// TIA Portal V20 export
ORGANIZATION_BLOCK "7000_Main"   // OB127, LAD, ProgramCycle
TITLE = "Main Program Sweep (Cycle)"
// stored: SetENOAutomatically false
   VAR_INPUT
      Initial_Call : Bool;   // Initial call of this OB
      Remanence : Bool;   // =True, if remanent data are available
   END_VAR
BEGIN

REGION Network 1: 2201_StackCalculate
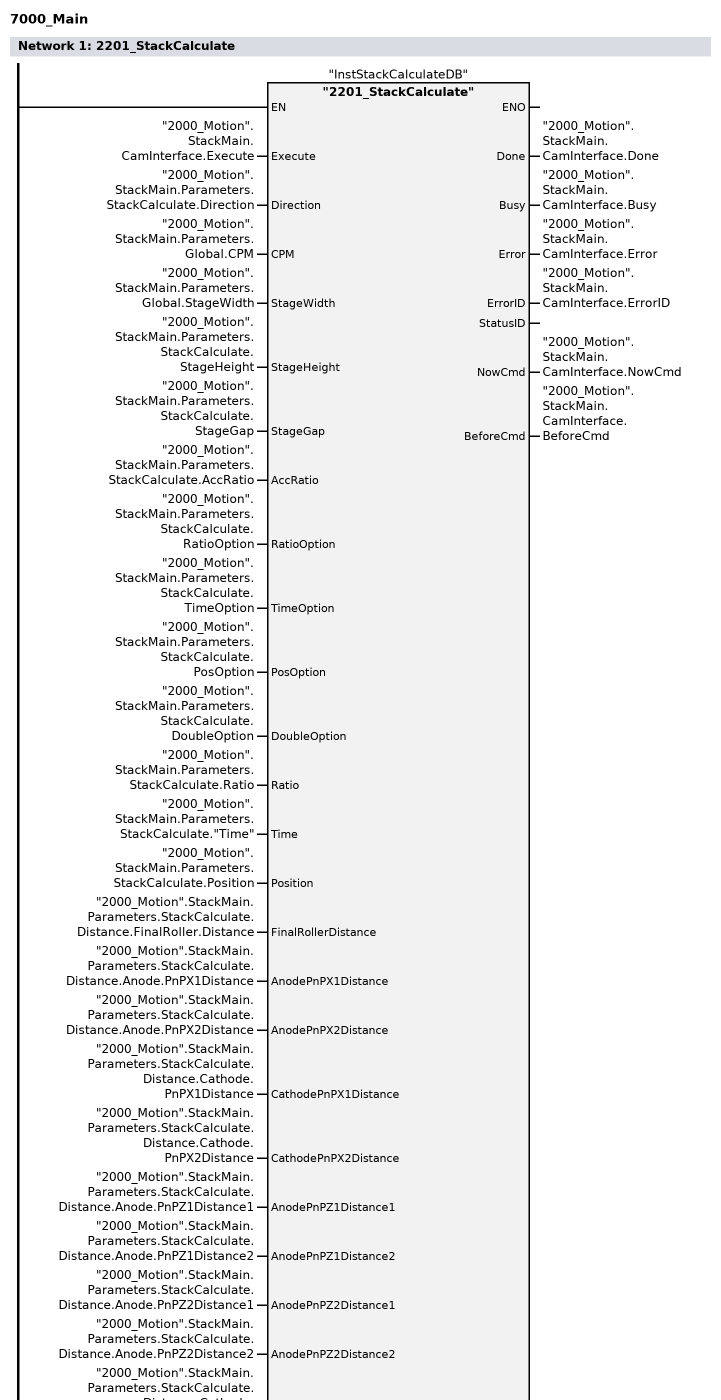
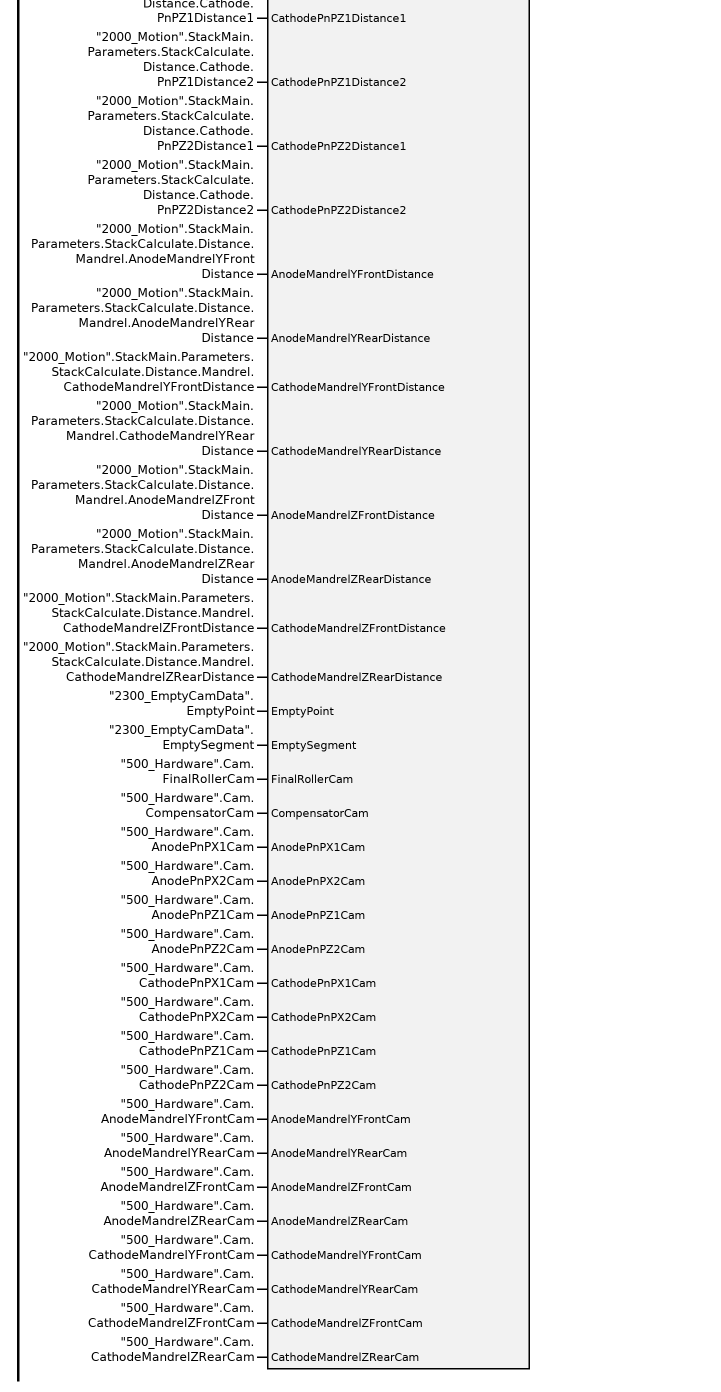
   RUNG wire#powerrail
      "InstStackCalculateDB"(Execute := "2000_Motion".StackMain.CamInterface.Execute, Direction := "2000_Motion".StackMain.Parameters.StackCalculate.Direction, CPM := "2000_Motion".StackMain.Parameters.Global.CPM, StageWidth := "2000_Motion".StackMain.Parameters.Global.StageWidth, StageHeight := "2000_Motion".StackMain.Parameters.StackCalculate.StageHeight, StageGap := "2000_Motion".StackMain.Parameters.StackCalculate.StageGap, AccRatio := "2000_Motion".StackMain.Parameters.StackCalculate.AccRatio, RatioOption := "2000_Motion".StackMain.Parameters.StackCalculate.RatioOption, TimeOption := "2000_Motion".StackMain.Parameters.StackCalculate.TimeOption, PosOption := "2000_Motion".StackMain.Parameters.StackCalculate.PosOption, DoubleOption := "2000_Motion".StackMain.Parameters.StackCalculate.DoubleOption, Ratio := "2000_Motion".StackMain.Parameters.StackCalculate.Ratio, "Time" := "2000_Motion".StackMain.Parameters.StackCalculate."Time", Position := "2000_Motion".StackMain.Parameters.StackCalculate.Position, FinalRollerDistance := "2000_Motion".StackMain.Parameters.StackCalculate.Distance.FinalRoller.Distance, AnodePnPX1Distance := "2000_Motion".StackMain.Parameters.StackCalculate.Distance.Anode.PnPX1Distance, AnodePnPX2Distance := "2000_Motion".StackMain.Parameters.StackCalculate.Distance.Anode.PnPX2Distance, CathodePnPX1Distance := "2000_Motion".StackMain.Parameters.StackCalculate.Distance.Cathode.PnPX1Distance, CathodePnPX2Distance := "2000_Motion".StackMain.Parameters.StackCalculate.Distance.Cathode.PnPX2Distance, AnodePnPZ1Distance1 := "2000_Motion".StackMain.Parameters.StackCalculate.Distance.Anode.PnPZ1Distance1, AnodePnPZ1Distance2 := "2000_Motion".StackMain.Parameters.StackCalculate.Distance.Anode.PnPZ1Distance2, AnodePnPZ2Distance1 := "2000_Motion".StackMain.Parameters.StackCalculate.Distance.Anode.PnPZ2Distance1, AnodePnPZ2Distance2 := "2000_Motion".StackMain.Parameters.StackCalculate.Distance.Anode.PnPZ2Distance2, CathodePnPZ1Distance1 := "2000_Motion".StackMain.Parameters.StackCalculate.Distance.Cathode.PnPZ1Distance1, CathodePnPZ1Distance2 := "2000_Motion".StackMain.Parameters.StackCalculate.Distance.Cathode.PnPZ1Distance2, CathodePnPZ2Distance1 := "2000_Motion".StackMain.Parameters.StackCalculate.Distance.Cathode.PnPZ2Distance1, CathodePnPZ2Distance2 := "2000_Motion".StackMain.Parameters.StackCalculate.Distance.Cathode.PnPZ2Distance2, AnodeMandrelYFrontDistance := "2000_Motion".StackMain.Parameters.StackCalculate.Distance.Mandrel.AnodeMandrelYFrontDistance, AnodeMandrelYRearDistance := "2000_Motion".StackMain.Parameters.StackCalculate.Distance.Mandrel.AnodeMandrelYRearDistance, CathodeMandrelYFrontDistance := "2000_Motion".StackMain.Parameters.StackCalculate.Distance.Mandrel.CathodeMandrelYFrontDistance, CathodeMandrelYRearDistance := "2000_Motion".StackMain.Parameters.StackCalculate.Distance.Mandrel.CathodeMandrelYRearDistance, AnodeMandrelZFrontDistance := "2000_Motion".StackMain.Parameters.StackCalculate.Distance.Mandrel.AnodeMandrelZFrontDistance, AnodeMandrelZRearDistance := "2000_Motion".StackMain.Parameters.StackCalculate.Distance.Mandrel.AnodeMandrelZRearDistance, CathodeMandrelZFrontDistance := "2000_Motion".StackMain.Parameters.StackCalculate.Distance.Mandrel.CathodeMandrelZFrontDistance, CathodeMandrelZRearDistance := "2000_Motion".StackMain.Parameters.StackCalculate.Distance.Mandrel.CathodeMandrelZRearDistance, EmptyPoint := "2300_EmptyCamData".EmptyPoint, EmptySegment := "2300_EmptyCamData".EmptySegment, FinalRollerCam := "500_Hardware".Cam.FinalRollerCam, CompensatorCam := "500_Hardware".Cam.CompensatorCam, AnodePnPX1Cam := "500_Hardware".Cam.AnodePnPX1Cam, AnodePnPX2Cam := "500_Hardware".Cam.AnodePnPX2Cam, AnodePnPZ1Cam := "500_Hardware".Cam.AnodePnPZ1Cam, AnodePnPZ2Cam := "500_Hardware".Cam.AnodePnPZ2Cam, CathodePnPX1Cam := "500_Hardware".Cam.CathodePnPX1Cam, CathodePnPX2Cam := "500_Hardware".Cam.CathodePnPX2Cam, CathodePnPZ1Cam := "500_Hardware".Cam.CathodePnPZ1Cam, CathodePnPZ2Cam := "500_Hardware".Cam.CathodePnPZ2Cam, AnodeMandrelYFrontCam := "500_Hardware".Cam.AnodeMandrelYFrontCam, AnodeMandrelYRearCam := "500_Hardware".Cam.AnodeMandrelYRearCam, AnodeMandrelZFrontCam := "500_Hardware".Cam.AnodeMandrelZFrontCam, AnodeMandrelZRearCam := "500_Hardware".Cam.AnodeMandrelZRearCam, CathodeMandrelYFrontCam := "500_Hardware".Cam.CathodeMandrelYFrontCam, CathodeMandrelYRearCam := "500_Hardware".Cam.CathodeMandrelYRearCam, CathodeMandrelZFrontCam := "500_Hardware".Cam.CathodeMandrelZFrontCam, CathodeMandrelZRearCam := "500_Hardware".Cam.CathodeMandrelZRearCam, Done => "2000_Motion".StackMain.CamInterface.Done, Busy => "2000_Motion".StackMain.CamInterface.Busy, Error => "2000_Motion".StackMain.CamInterface.Error, ErrorID => "2000_Motion".StackMain.CamInterface.ErrorID, NowCmd => "2000_Motion".StackMain.CamInterface.NowCmd, BeforeCmd => "2000_Motion".StackMain.CamInterface.BeforeCmd, StatusID =>)
   END_RUNG
   // the same network as SCL:
   "InstStackCalculateDB"(Execute := "2000_Motion".StackMain.CamInterface.Execute,   // "2201_StackCalculate"
                          Direction := "2000_Motion".StackMain.Parameters.StackCalculate.Direction,
                          CPM := "2000_Motion".StackMain.Parameters.Global.CPM,
                          StageWidth := "2000_Motion".StackMain.Parameters.Global.StageWidth,
                          StageHeight := "2000_Motion".StackMain.Parameters.StackCalculate.StageHeight,
                          StageGap := "2000_Motion".StackMain.Parameters.StackCalculate.StageGap,
                          AccRatio := "2000_Motion".StackMain.Parameters.StackCalculate.AccRatio,
                          RatioOption := "2000_Motion".StackMain.Parameters.StackCalculate.RatioOption,
                          TimeOption := "2000_Motion".StackMain.Parameters.StackCalculate.TimeOption,
                          PosOption := "2000_Motion".StackMain.Parameters.StackCalculate.PosOption,
                          DoubleOption := "2000_Motion".StackMain.Parameters.StackCalculate.DoubleOption,
                          Ratio := "2000_Motion".StackMain.Parameters.StackCalculate.Ratio,
                          "Time" := "2000_Motion".StackMain.Parameters.StackCalculate."Time",
                          Position := "2000_Motion".StackMain.Parameters.StackCalculate.Position,
                          FinalRollerDistance := "2000_Motion".StackMain.Parameters.StackCalculate.Distance.FinalRoller.Distance,
                          AnodePnPX1Distance := "2000_Motion".StackMain.Parameters.StackCalculate.Distance.Anode.PnPX1Distance,
                          AnodePnPX2Distance := "2000_Motion".StackMain.Parameters.StackCalculate.Distance.Anode.PnPX2Distance,
                          CathodePnPX1Distance := "2000_Motion".StackMain.Parameters.StackCalculate.Distance.Cathode.PnPX1Distance,
                          CathodePnPX2Distance := "2000_Motion".StackMain.Parameters.StackCalculate.Distance.Cathode.PnPX2Distance,
                          AnodePnPZ1Distance1 := "2000_Motion".StackMain.Parameters.StackCalculate.Distance.Anode.PnPZ1Distance1,
                          AnodePnPZ1Distance2 := "2000_Motion".StackMain.Parameters.StackCalculate.Distance.Anode.PnPZ1Distance2,
                          AnodePnPZ2Distance1 := "2000_Motion".StackMain.Parameters.StackCalculate.Distance.Anode.PnPZ2Distance1,
                          AnodePnPZ2Distance2 := "2000_Motion".StackMain.Parameters.StackCalculate.Distance.Anode.PnPZ2Distance2,
                          CathodePnPZ1Distance1 := "2000_Motion".StackMain.Parameters.StackCalculate.Distance.Cathode.PnPZ1Distance1,
                          CathodePnPZ1Distance2 := "2000_Motion".StackMain.Parameters.StackCalculate.Distance.Cathode.PnPZ1Distance2,
                          CathodePnPZ2Distance1 := "2000_Motion".StackMain.Parameters.StackCalculate.Distance.Cathode.PnPZ2Distance1,
                          CathodePnPZ2Distance2 := "2000_Motion".StackMain.Parameters.StackCalculate.Distance.Cathode.PnPZ2Distance2,
                          AnodeMandrelYFrontDistance := "2000_Motion".StackMain.Parameters.StackCalculate.Distance.Mandrel.AnodeMandrelYFrontDistance,
                          AnodeMandrelYRearDistance := "2000_Motion".StackMain.Parameters.StackCalculate.Distance.Mandrel.AnodeMandrelYRearDistance,
                          CathodeMandrelYFrontDistance := "2000_Motion".StackMain.Parameters.StackCalculate.Distance.Mandrel.CathodeMandrelYFrontDistance,
                          CathodeMandrelYRearDistance := "2000_Motion".StackMain.Parameters.StackCalculate.Distance.Mandrel.CathodeMandrelYRearDistance,
                          AnodeMandrelZFrontDistance := "2000_Motion".StackMain.Parameters.StackCalculate.Distance.Mandrel.AnodeMandrelZFrontDistance,
                          AnodeMandrelZRearDistance := "2000_Motion".StackMain.Parameters.StackCalculate.Distance.Mandrel.AnodeMandrelZRearDistance,
                          CathodeMandrelZFrontDistance := "2000_Motion".StackMain.Parameters.StackCalculate.Distance.Mandrel.CathodeMandrelZFrontDistance,
                          CathodeMandrelZRearDistance := "2000_Motion".StackMain.Parameters.StackCalculate.Distance.Mandrel.CathodeMandrelZRearDistance,
                          EmptyPoint := "2300_EmptyCamData".EmptyPoint,
                          EmptySegment := "2300_EmptyCamData".EmptySegment,
                          FinalRollerCam := "500_Hardware".Cam.FinalRollerCam,
                          CompensatorCam := "500_Hardware".Cam.CompensatorCam,
                          AnodePnPX1Cam := "500_Hardware".Cam.AnodePnPX1Cam,
                          AnodePnPX2Cam := "500_Hardware".Cam.AnodePnPX2Cam,
                          AnodePnPZ1Cam := "500_Hardware".Cam.AnodePnPZ1Cam,
                          AnodePnPZ2Cam := "500_Hardware".Cam.AnodePnPZ2Cam,
                          CathodePnPX1Cam := "500_Hardware".Cam.CathodePnPX1Cam,
                          CathodePnPX2Cam := "500_Hardware".Cam.CathodePnPX2Cam,
                          CathodePnPZ1Cam := "500_Hardware".Cam.CathodePnPZ1Cam,
                          CathodePnPZ2Cam := "500_Hardware".Cam.CathodePnPZ2Cam,
                          AnodeMandrelYFrontCam := "500_Hardware".Cam.AnodeMandrelYFrontCam,
                          AnodeMandrelYRearCam := "500_Hardware".Cam.AnodeMandrelYRearCam,
                          AnodeMandrelZFrontCam := "500_Hardware".Cam.AnodeMandrelZFrontCam,
                          AnodeMandrelZRearCam := "500_Hardware".Cam.AnodeMandrelZRearCam,
                          CathodeMandrelYFrontCam := "500_Hardware".Cam.CathodeMandrelYFrontCam,
                          CathodeMandrelYRearCam := "500_Hardware".Cam.CathodeMandrelYRearCam,
                          CathodeMandrelZFrontCam := "500_Hardware".Cam.CathodeMandrelZFrontCam,
                          CathodeMandrelZRearCam := "500_Hardware".Cam.CathodeMandrelZRearCam,
                          Done => "2000_Motion".StackMain.CamInterface.Done,
                          Busy => "2000_Motion".StackMain.CamInterface.Busy,
                          Error => "2000_Motion".StackMain.CamInterface.Error,
                          ErrorID => "2000_Motion".StackMain.CamInterface.ErrorID,
                          NowCmd => "2000_Motion".StackMain.CamInterface.NowCmd,
                          BeforeCmd => "2000_Motion".StackMain.CamInterface.BeforeCmd);
END_REGION
END_ORGANIZATION_BLOCK
